// TwinCAT 3 PLC project Untitled1
// ProgramVersion: 3.1.4020.2
// libraries:
//   Tc2_Standard, * (Beckhoff Automation GmbH)
//   Tc2_System, * (Beckhoff Automation GmbH)
//   Tc3_Module, * (Beckhoff Automation GmbH)
// project tree:
//   DUTs/ ST_Record.TcDUT
//   / PlcTask.TcTTO
//   POUs/ MAIN.TcPOU
// real-time tasks:
//   TASK PlcTask: cycle T#10ms, priority 20, ADS port 350

CONFIGURATION Untitled1
    RESOURCE PLC ON TwinCAT3
        TASK PlcTask(INTERVAL := T#10ms, PRIORITY := 20);
        PROGRAM MAIN WITH PlcTask : MAIN;
    END_RESOURCE
END_CONFIGURATION

// ---- DUTs/ST_Record.TcDUT
TYPE ST_Record :
STRUCT
	test : ARRAY[0..99999] OF DWORD;
	test2 : ARRAY[0..99999] OF DWORD;
	test3 : ARRAY[0..99999] OF DWORD;
END_STRUCT
END_TYPE

// ---- POUs/MAIN.TcPOU
PROGRAM MAIN
VAR
	record : ST_Record;
	bla : DWORD;
END_VAR

bla := record.test[9999];

END_PROGRAM
